INTERFACE ITF_MCHMIPrepareScreen_06_XX_Init

METHOD PUBLIC LinkDataHMI_06_XX : BOOL
VAR_INPUT
	refstData				: REFERENCE TO ST_MCHMIPrepareScreen_06_XX;
END_VAR
END_METHOD

END_INTERFACE

(* stored: Version 1.1.0.1
   Itf ITF_MCHMIPrepareScreen_06_XX_Init: Id {3b32dd81-f8ae-0512-02ef-3ea1bdee3165}
   Method LinkDataHMI_06_XX: Id {7d106f31-48e9-0dd9-37f4-24ff3b7f6f76} *)
